{attribute 'qualified_only'}
VAR_GLOBAL
	i_TasterYellow AT%I* : BOOL;
END_VAR

(* stored: Version 1.1.0.1, ProductVersion 3.1.4022.12
   GVL GVL: Id {79a3af6f-de66-4038-b2af-a00018d839a3} *)
